(* IEC 61131-3 sources: Industry-PLC-LLM/data/PLCBEAD_repo/PLCBEAD_PLCEmbed-main/PLC-BEAD/Source/GEB/_REAL_TO_UDINT, 1 file *)

(* ---- _REAL_TO_UDINT.ST ---- *)
FUNCTION _REAL_TO_UDINT:UDINT
  VAR_INPUT
    X :	REAL;
  END_VAR

  IF REAL_TO_UDINT(0.5) = UDINT#1 THEN
    _REAL_TO_UDINT := REAL_TO_UDINT(X);
  ELSIF X > 0.0 THEN
    _REAL_TO_UDINT := REAL_TO_UDINT(X+0.5);
  ELSIF X < 0.0 THEN
    _REAL_TO_UDINT := REAL_TO_UDINT(X-0.5);
  ELSE
    _REAL_TO_UDINT := UDINT#0;
  END_IF;
END_FUNCTION

PROGRAM program0
    VAR
      LocalVar0 : REAL;
      LocalOUT  : UDINT;
    END_VAR

    LocalOUT := _REAL_TO_UDINT(LocalVar0);
END_PROGRAM
